PROGRAM MAIN
VAR
	fbMachine				: FB_Machine;
END_VAR

fbMachine();

END_PROGRAM

(* stored: Version 1.1.0.1, ProductVersion 3.1.4024.12
   POU MAIN: Id {04ba039b-795a-46fa-8d67-a13d131c6641}, SpecialFunc None *)
